Yaskawa INFORM job: long_pipe.JBI

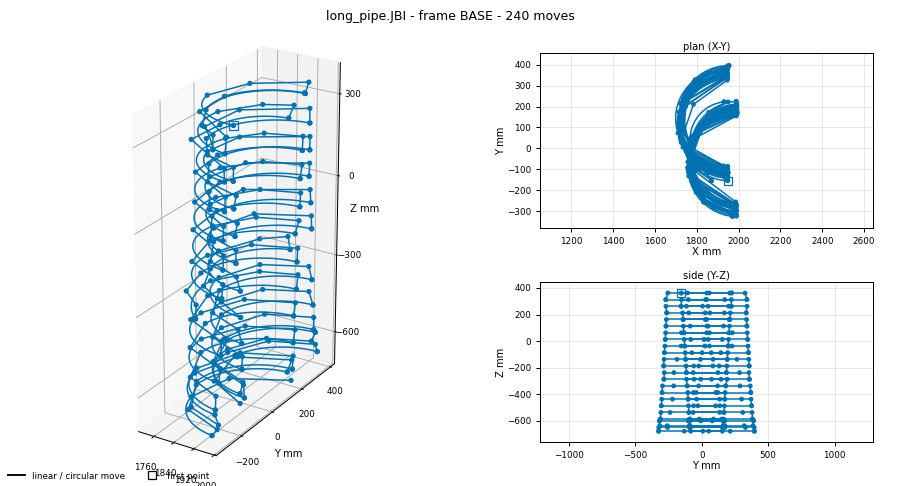
[picture p0: tool path of long_pipe.JBI in frame BASE, 240 of 346 moves have a stored position in this frame; points joined in program order, loops and branches not executed]
/JOB
//NAME long_pipe
//POS
///NPOS 336,0,336,0,0,0
///TOOL 0
///POSTYPE BASE
///RECTAN
///RCONF 0,0,0,0,0,0,0,0,0,0,0,0,0,0,0,0,0,0,0,0,0,0,0,0
C00000=1948.089852,-154.428104,361.796500,-91.436421,-90.000000,5.000000
C00001=1948.089852,-154.428104,361.796500,-91.436421,-90.000000,5.000000
C00002=1806.657138,-101.141800,361.796500,-121.772810,-90.000000,5.000000
C00003=1725.085960,37.670682,361.796500,-156.237975,-90.000000,5.000000
C00004=1725.085960,37.670682,361.796500,-156.237975,-90.000000,5.000000
C00005=1784.341244,210.221855,361.796500,157.427074,-90.000000,5.000000
C00006=1945.915028,325.931055,361.796500,92.921430,-89.999999,5.000000
C00007=1924.685573,339.998740,312.680000,98.705914,-90.000000,5.000000
C00008=1924.685573,339.998740,312.680000,98.705914,-90.000000,5.000000
C00009=1721.013871,191.051148,312.680000,167.503050,-90.000000,5.000000
C00010=1725.983821,28.850345,312.680000,-154.339335,-90.000000,5.000000
C00011=1725.983821,28.850345,312.680000,-154.339335,-90.000000,5.000000
C00012=1795.223122,-101.158175,312.680000,-123.700098,-90.000000,5.000000
C00013=1869.864544,-152.794566,312.680000,-106.341970,-90.000000,5.000000
C00014=1870.472685,-155.549095,262.680000,-106.088120,-90.000000,5.000000
C00015=1870.472685,-155.549095,262.680000,-106.088120,-90.000000,5.000000
C00016=1843.579568,-119.383824,262.680000,-113.403433,-90.000000,5.000000
C00017=1734.255940,6.180166,262.680000,-148.999232,-90.000000,5.000000
C00018=1734.255940,6.180166,262.680000,-148.999232,-90.000000,5.000000
C00019=1747.769146,201.411479,262.680000,163.296650,-90.000000,5.000000
C00020=1942.694355,340.824041,262.680000,93.618014,-90.000000,5.000000
C00021=1947.073941,334.429289,212.680000,92.455325,-90.000000,5.000000
C00022=1947.073941,334.429289,212.680000,92.455325,-90.000000,5.000000
C00023=1743.822934,197.595389,212.680000,164.546518,-90.000000,5.000000
C00024=1728.032875,25.819450,212.680000,-153.523098,-90.000000,5.000000
C00025=1728.032875,25.819450,212.680000,-153.523098,-90.000000,5.000000
C00026=1812.698059,-97.501858,212.680000,-121.105327,-90.000000,5.000000
C00027=1942.399423,-144.705270,212.680000,-92.632933,-90.000000,5.000000
C00028=1938.946956,-141.309317,162.680000,-93.368274,-90.000000,5.000000
C00029=1938.946956,-141.309317,162.680000,-93.368274,-90.000000,5.000000
C00030=1803.563456,-88.140401,162.680000,-123.759652,-89.999999,5.000000
C00031=1725.441837,36.442533,162.680000,-155.949661,-90.000000,5.000000
C00032=1725.441837,36.442533,162.680000,-155.949661,-90.000000,5.000000
C00033=1746.336332,205.754669,162.680000,162.318158,-90.000000,5.000000
C00034=1946.808055,337.053275,162.680000,92.499632,-90.000000,5.000000
C00035=1945.260351,339.688853,112.680000,92.907920,-89.999999,5.000000
C00036=1945.260351,339.688853,112.680000,92.907920,-89.999999,5.000000
C00037=1749.833887,217.231411,112.680000,159.191678,-90.000000,5.000000
C00038=1723.055881,48.584757,112.680000,-158.721498,-90.000000,5.000000
C00039=1723.055881,48.584757,112.680000,-158.721498,-90.000000,5.000000
C00040=1805.768560,-87.049483,112.680000,-123.500409,-90.000000,5.000000
C00041=1949.000324,-138.863334,112.680000,-91.329258,-90.000000,5.000000
C00042=1936.884281,-134.495510,62.680000,-93.882169,-90.000000,5.000000
C00043=1936.884281,-134.495510,62.680000,-93.882169,-90.000000,5.000000
C00044=1804.163203,-80.705374,62.680000,-124.539805,-89.999999,5.000000
C00045=1721.098993,58.361092,62.680000,-160.992048,-89.999999,5.000000
C00046=1721.098993,58.361092,62.680000,-160.992048,-89.999999,5.000000
C00047=1755.943683,229.421087,62.680000,155.640501,-90.000000,5.000000
C00048=1943.839534,342.441100,62.680000,93.267809,-89.999999,5.000000
C00049=1940.731812,345.123724,12.680000,94.086050,-90.000000,5.000000
C00050=1940.731812,345.123724,12.680000,94.086050,-90.000000,5.000000
C00051=1755.079974,233.890953,12.680000,154.680026,-90.000000,5.000000
C00052=1723.758836,48.110633,12.680000,-158.561082,-90.000000,5.000000
C00053=1723.758836,48.110633,12.680000,-158.561082,-90.000000,5.000000
C00054=1810.808406,-83.344167,12.680000,-123.034502,-89.999999,5.000000
C00055=1949.054836,-132.185836,12.680000,-91.350458,-90.000000,5.000000
C00056=1937.608440,-128.432526,-37.320000,-93.815495,-90.000000,5.000000
C00057=1937.608440,-128.432526,-37.320000,-93.815495,-90.000000,5.000000
C00058=1801.716874,-73.293020,-37.320000,-125.898714,-90.000000,5.000000
C00059=1721.874769,57.373947,-37.320000,-160.717445,-90.000000,5.000000
C00060=1721.874769,57.373947,-37.320000,-160.717445,-90.000000,5.000000
C00061=1748.048392,227.228459,-37.320000,156.976432,-90.000000,5.000000
C00062=1943.886424,348.166100,-37.320000,93.165704,-90.000000,5.000000
C00063=1945.403570,351.508515,-87.320000,92.707825,-90.000000,5.000000
C00064=1945.403570,351.508515,-87.320000,92.707825,-90.000000,5.000000
C00065=1764.794043,254.451315,-87.320000,148.823101,-90.000000,5.000000
C00066=1719.364469,71.495201,-87.320000,-164.022571,-90.000000,5.000000
C00067=1719.364469,71.495201,-87.320000,-164.022571,-90.000000,5.000000
C00068=1809.133318,-75.149384,-87.320000,-124.331343,-89.999999,5.000000
C00069=1938.729832,-125.214955,-87.320000,-93.619745,-89.999999,5.000000
C00070=1936.922427,-121.754242,-137.320000,-94.062838,-90.000000,5.000000
C00071=1936.922427,-121.754242,-137.320000,-94.062838,-90.000000,5.000000
C00072=1805.471154,-68.553083,-137.320000,-125.840133,-90.000000,5.000000
C00073=1717.543155,84.697835,-137.320000,-167.121689,-89.999999,5.000000
C00074=1717.543155,84.697835,-137.320000,-167.121689,-89.999999,5.000000
C00075=1769.057610,264.695420,-137.320000,146.025114,-90.000000,5.000000
C00076=1946.343505,354.471103,-137.320000,92.421083,-90.000000,5.000000
C00077=1946.850856,357.205562,-187.320000,92.257711,-90.000000,5.000000
C00078=1946.850856,357.205562,-187.320000,92.257711,-90.000000,5.000000
C00079=1769.073697,266.901665,-187.320000,145.558968,-90.000000,5.000000
C00080=1718.050928,83.425907,-187.320000,-166.803742,-90.000000,5.000000
C00081=1718.050928,83.425907,-187.320000,-166.803742,-90.000000,5.000000
C00082=1796.817162,-60.318135,-187.320000,-128.502754,-90.000000,5.000000
C00083=1936.521124,-118.597040,-187.320000,-94.201205,-90.000000,5.000000
C00084=1950.373259,-115.822362,-237.320000,-91.140926,-90.000000,5.000000
C00085=1950.373259,-115.822362,-237.320000,-91.140926,-90.000000,5.000000
C00086=1788.789474,-49.698601,-237.320000,-131.437564,-90.000000,5.000000
C00087=1713.556771,121.462071,-237.320000,-175.831712,-89.999999,5.000000
C00088=1713.556771,121.462071,-237.320000,-175.831712,-89.999999,5.000000
C00089=1779.676107,284.296664,-237.320000,140.440110,-89.999999,5.000000
C00090=1853.162637,354.889370,-237.320000,115.360721,-89.999999,5.000000
C00091=1860.386180,358.675829,-287.320000,113.409006,-90.000000,5.000000
C00092=1860.386180,358.675829,-287.320000,113.409006,-90.000000,5.000000
C00093=1730.946298,258.659756,-287.320000,151.960616,-89.999999,5.000000
C00094=1710.739488,73.262255,-287.320000,-164.943488,-89.999999,5.000000
C00095=1710.739488,73.262255,-287.320000,-164.943488,-89.999999,5.000000
C00096=1767.064394,-57.558684,-287.320000,-133.770440,-90.000000,5.000000
C00097=1859.771689,-115.665984,-287.320000,-110.584520,-90.000000,5.000000
C00098=1947.779730,-109.811027,-337.320000,-91.765092,-90.000000,5.000000
C00099=1947.779730,-109.811027,-337.320000,-91.765092,-90.000000,5.000000
C00100=1794.208585,-45.495626,-337.320000,-131.138093,-90.000000,5.000000
C00101=1715.967037,119.350089,-337.320000,-175.287684,-89.999999,5.000000
C00102=1715.967037,119.350089,-337.320000,-175.287684,-89.999999,5.000000
C00103=1779.362251,288.057746,-337.320000,139.769441,-89.999999,5.000000
C00104=1933.415288,364.951223,-337.320000,95.572089,-90.000000,5.000000
C00105=1944.191004,368.935356,-387.320000,92.804410,-90.000000,5.000000
C00106=1944.191004,368.935356,-387.320000,92.804410,-90.000000,5.000000
C00107=1776.821526,289.635713,-387.320000,139.876442,-90.000000,5.000000
C00108=1716.129048,121.164597,-387.320000,-175.716243,-89.999999,5.000000
C00109=1716.129048,121.164597,-387.320000,-175.716243,-89.999999,5.000000
C00110=1793.249925,-42.090790,-387.320000,-131.835982,-90.000000,5.000000
C00111=1934.966448,-105.589525,-387.320000,-94.785386,-89.999999,5.000000
C00112=1947.760101,-102.612541,-437.320000,-91.822275,-90.000000,5.000000
C00113=1947.760101,-102.612541,-437.320000,-91.822275,-90.000000,5.000000
C00114=1789.178214,-35.129272,-437.320000,-133.662724,-90.000000,5.000000
C00115=1715.792418,134.107597,-437.320000,-178.808772,-90.000000,5.000000
C00116=1715.792418,134.107597,-437.320000,-178.808772,-90.000000,5.000000
C00117=1783.843259,300.141568,-437.320000,136.817550,-90.000000,5.000000
C00118=1931.738733,371.088649,-437.320000,95.835639,-90.000000,5.000000
C00119=1946.586127,374.922161,-487.320000,92.152487,-89.999999,5.000000
C00120=1946.586127,374.922161,-487.320000,92.152487,-89.999999,5.000000
C00121=1781.433288,301.447997,-487.320000,136.985248,-90.000000,5.000000
C00122=1715.605097,135.687903,-487.320000,-179.187100,-90.000000,5.000000
C00123=1715.605097,135.687903,-487.320000,-179.187100,-90.000000,5.000000
C00124=1784.593790,-28.973026,-487.320000,-135.472019,-90.000000,5.000000
C00125=1948.352074,-100.171239,-487.320000,-91.699232,-90.000000,5.000000
C00126=1945.281183,-97.217812,-537.320000,-92.464026,-89.999999,5.000000
C00127=1945.281183,-97.217812,-537.320000,-92.464026,-89.999999,5.000000
C00128=1793.117537,-33.362696,-537.320000,-133.268365,-90.000000,5.000000
C00129=1716.145427,134.684238,-537.320000,-178.945025,-89.999999,5.000000
C00130=1716.145427,134.684238,-537.320000,-178.945025,-89.999999,5.000000
C00131=1787.067288,308.692942,-537.320000,134.793315,-90.000000,5.000000
C00132=1948.021952,378.690968,-537.320000,91.775708,-90.000000,5.000000
C00133=1947.011560,381.966547,-587.320000,91.989878,-90.000000,5.000000
C00134=1947.011560,381.966547,-587.320000,91.989878,-90.000000,5.000000
C00135=1789.216558,315.135500,-587.320000,133.358123,-90.000000,5.000000
C00136=1716.024354,149.961106,-587.320000,177.400513,-89.999999,5.000000
C00137=1716.024354,149.961106,-587.320000,177.400513,-89.999999,5.000000
C00138=1778.857613,-18.448199,-587.320000,-138.263643,-90.000000,5.000000
C00139=1947.332074,-94.134217,-587.320000,-91.993503,-90.000000,5.000000
C00140=1933.662341,-90.882022,-637.320000,-95.412052,-90.000000,5.000000
C00141=1933.662341,-90.882022,-637.320000,-95.412052,-90.000000,5.000000
C00142=1767.208531,-2.444827,-637.320000,-143.061065,-90.000000,5.000000
C00143=1716.921361,173.665472,-637.320000,171.752478,-89.999999,5.000000
C00144=1716.921361,173.665472,-637.320000,171.752478,-89.999999,5.000000
C00145=1789.055258,319.507135,-637.320000,132.684821,-90.000000,5.000000
C00146=1936.254340,385.591245,-637.320000,94.452796,-90.000000,5.000000
C00147=1949.256140,389.855264,-600.717460,180.000000,-60.000000,-88.585086
C00148=1949.256140,389.855264,-600.717460,180.000000,-60.000000,-88.585086
C00149=1796.012674,328.533492,-600.717460,180.000000,-60.000000,-49.915588
C00150=1716.317998,172.325490,-600.717460,180.000000,-60.000000,-7.912266
C00151=1716.317998,172.325490,-600.717460,180.000000,-60.000000,-7.912266
C00152=1775.299054,-8.028706,-600.717460,180.000000,-60.000000,39.236687
C00153=1946.064111,-89.050219,-600.717460,180.000000,-60.000000,87.644140
C00154=1948.372494,-86.795927,-650.717460,180.000000,-60.000000,88.205392
C00155=1948.372494,-86.795927,-650.717460,180.000000,-60.000000,88.205392
C00156=1775.279847,-6.023758,-650.717460,180.000000,-60.000000,38.849071
C00157=1716.545205,174.101681,-650.717460,180.000000,-60.000000,-8.337156
C00158=1716.545205,174.101681,-650.717460,180.000000,-60.000000,-8.337156
C00159=1792.571085,328.575973,-650.717460,-180.000000,-60.000000,-49.318058
C00160=1947.362979,394.502867,-650.717460,-180.000000,-60.000000,-88.186469
C00161=1954.969684,396.112738,-678.637460,-180.000000,-60.000000,-89.892927
C00162=1954.969684,396.112738,-678.637460,-180.000000,-60.000000,-89.892927
C00163=1803.482227,342.074602,-678.637460,-180.000000,-60.000000,-53.178896
C00164=1721.591344,214.572083,-678.637460,180.000000,-60.000000,-17.888195
C00165=1721.591344,214.572083,-678.637460,180.000000,-60.000000,-17.888195
C00166=1765.108221,8.381083,-678.637460,180.000000,-60.000000,34.477840
C00167=1929.576251,-83.832453,-678.637460,180.000000,-60.000000,83.379552
C00168=1988.723901,224.495613,362.682500,91.136861,-90.000000,5.000000
C00169=1988.723901,224.495613,362.682500,91.136861,-90.000000,5.000000
C00170=1851.653962,169.776784,362.682500,120.888805,-90.000000,5.000000
C00171=1780.186310,57.522696,362.682500,149.431820,-90.000000,5.000000
C00172=1780.186310,57.522696,362.682500,149.431820,-90.000000,5.000000
C00173=1789.875186,-107.742667,362.682500,-169.305957,-89.999999,5.000000
C00174=1986.239805,-255.786622,362.682500,-92.548667,-89.999999,5.000000
C00175=1990.121191,-271.036941,312.680000,-91.256333,-90.000000,5.000000
C00176=1990.121191,-271.036941,312.680000,-91.256333,-90.000000,5.000000
C00177=1808.253351,-148.428142,312.680000,-156.932564,-89.999999,5.000000
C00178=1767.408881,36.499458,312.680000,155.067828,-90.000000,5.000000
C00179=1767.408881,36.499458,312.680000,155.067828,-90.000000,5.000000
C00180=1857.792979,173.043612,312.680000,119.457652,-90.000000,5.000000
C00181=1950.206892,222.480952,312.680000,98.647445,-90.000000,5.000000
C00182=1930.045697,222.355400,262.680000,102.479797,-89.999999,5.000000
C00183=1930.045697,222.355400,262.680000,102.479797,-89.999999,5.000000
C00184=1817.772394,166.172520,262.680000,126.921293,-90.000000,5.000000
C00185=1768.075189,47.416654,262.680000,152.776908,-89.999999,5.000000
C00186=1768.075189,47.416654,262.680000,152.776908,-89.999999,5.000000
C00187=1760.588722,-115.433226,262.680000,-168.796077,-90.000000,5.000000
C00188=1985.937756,-270.370881,262.680000,-92.450043,-89.999999,5.000000
C00189=1983.203786,-264.021545,212.680000,-93.331225,-90.000000,5.000000
C00190=1983.203786,-264.021545,212.680000,-93.331225,-90.000000,5.000000
C00191=1778.387774,-96.104856,212.680000,-172.876660,-90.000000,5.000000
C00192=1781.359778,60.338071,212.680000,148.737810,-90.000000,5.000000
C00193=1781.359778,60.338071,212.680000,148.737810,-90.000000,5.000000
C00194=1865.910821,170.095672,212.680000,118.272216,-89.999999,5.000000
C00195=1990.964908,214.652948,212.680000,90.723891,-89.999999,5.000000
C00196=1990.361250,211.531002,162.680000,90.855171,-90.000000,5.000000
C00197=1990.361250,211.531002,162.680000,90.855171,-90.000000,5.000000
C00198=1855.009552,160.725264,162.680000,121.265397,-90.000000,5.000000
C00199=1771.949454,26.848917,162.680000,156.684157,-89.999999,5.000000
C00200=1771.949454,26.848917,162.680000,156.684157,-89.999999,5.000000
C00201=1792.474616,-139.695411,162.680000,-160.740769,-89.999999,5.000000
C00202=1988.687598,-266.951202,162.680000,-91.697121,-89.999999,5.000000
C00203=1986.544852,-269.556546,112.680000,-92.286765,-90.000000,5.000000
C00204=1986.544852,-269.556546,112.680000,-92.286765,-90.000000,5.000000
C00205=1788.365526,-135.956463,112.680000,-162.032162,-89.999999,5.000000
C00206=1774.573122,38.290928,112.680000,153.980638,-89.999999,5.000000
C00207=1774.573122,38.290928,112.680000,153.980638,-89.999999,5.000000
C00208=1865.058629,163.596407,112.680000,119.096094,-90.000000,5.000000
C00209=1991.745006,208.618149,112.680000,90.578695,-90.000000,5.000000
C00210=1987.652745,204.721634,62.680000,91.442958,-89.999999,5.000000
C00211=1987.652745,204.721634,62.680000,91.442958,-89.999999,5.000000
C00212=1860.097116,157.587789,62.680000,120.673992,-90.000000,5.000000
C00213=1774.256284,36.753283,62.680000,154.337162,-90.000000,5.000000
C00214=1774.256284,36.753283,62.680000,154.337162,-90.000000,5.000000
C00215=1797.219859,-153.509246,62.680000,-156.838660,-90.000000,5.000000
C00216=1985.392353,-272.459154,62.680000,-92.578281,-90.000000,5.000000
C00217=1983.896404,-274.918472,12.680000,-92.962976,-90.000000,5.000000
C00218=1983.896404,-274.918472,12.680000,-92.962976,-90.000000,5.000000
C00219=1802.598281,-166.501797,12.680000,-153.093322,-90.000000,5.000000
C00220=1769.911825,17.517256,12.680000,158.916075,-90.000000,5.000000
C00221=1769.911825,17.517256,12.680000,158.916075,-90.000000,5.000000
C00222=1860.434601,154.194398,12.680000,120.990949,-90.000000,5.000000
C00223=1991.728115,201.901968,12.680000,90.596607,-90.000000,5.000000
C00224=1990.844367,198.678738,-37.320000,90.792859,-89.999999,5.000000
C00225=1990.844367,198.678738,-37.320000,90.792859,-89.999999,5.000000
C00226=1848.887250,145.095727,-37.320000,124.218588,-90.000000,5.000000
C00227=1770.707112,23.440533,-37.320000,157.540917,-90.000000,5.000000
C00228=1770.707112,23.440533,-37.320000,157.540917,-90.000000,5.000000
C00229=1791.125725,-155.813653,-37.320000,-156.910761,-89.999999,5.000000
C00230=1987.626168,-278.204845,-37.320000,-91.896390,-90.000000,5.000000
C00231=1987.302870,-281.404691,-87.320000,-91.954979,-90.000000,5.000000
C00232=1987.302870,-281.404691,-87.320000,-91.954979,-90.000000,5.000000
C00233=1802.163860,-174.716993,-87.320000,-151.231840,-90.000000,5.000000
C00234=1766.018401,2.495406,-87.320000,162.607090,-90.000000,5.000000
C00235=1766.018401,2.495406,-87.320000,162.607090,-90.000000,5.000000
C00236=1852.133956,143.567440,-87.320000,123.809976,-90.000000,5.000000
C00237=1990.301803,195.483467,-87.320000,90.919903,-90.000000,5.000000
C00238=1978.075101,191.483388,-137.320000,93.617729,-90.000000,5.000000
C00239=1978.075101,191.483388,-137.320000,93.617729,-90.000000,5.000000
C00240=1840.480246,132.727671,-137.320000,127.358362,-89.999999,5.000000
C00241=1763.569258,-10.937979,-137.320000,165.868582,-90.000000,5.000000
C00242=1763.569258,-10.937979,-137.320000,165.868582,-90.000000,5.000000
C00243=1805.736775,-186.129334,-137.320000,-148.206757,-90.000000,5.000000
C00244=1988.495735,-284.497788,-137.320000,-91.609942,-90.000000,5.000000
C00245=1986.431281,-287.235224,-187.320000,-92.131405,-90.000000,5.000000
C00246=1986.431281,-287.235224,-187.320000,-92.131405,-90.000000,5.000000
C00247=1811.881725,-196.821195,-187.320000,-145.036956,-90.000000,5.000000
C00248=1761.960998,-22.671143,-187.320000,168.713269,-90.000000,5.000000
C00249=1761.960998,-22.671143,-187.320000,168.713269,-90.000000,5.000000
C00250=1841.420154,130.973540,-187.320000,127.430524,-89.999999,5.000000
C00251=1990.349923,189.068152,-187.320000,90.932082,-90.000000,5.000000
C00252=1990.050783,185.617204,-237.320000,91.011979,-90.000000,5.000000
C00253=1990.050783,185.617204,-237.320000,91.011979,-90.000000,5.000000
C00254=1834.684708,121.001254,-237.320000,130.063431,-89.999999,5.000000
C00255=1760.682694,-64.207382,-237.320000,178.803723,-90.000000,5.000000
C00256=1760.682694,-64.207382,-237.320000,178.803723,-90.000000,5.000000
C00257=1797.351101,-209.746240,-237.320000,-144.501034,-90.000000,5.000000
C00258=1883.887097,-282.491417,-237.320000,-117.409868,-90.000000,5.000000
C00259=1883.201806,-285.218759,-287.320000,-117.257350,-90.000000,5.000000
C00260=1883.201806,-285.218759,-287.320000,-117.257350,-90.000000,5.000000
C00261=1825.084107,-222.094242,-287.320000,-137.922519,-89.999999,5.000000
C00262=1764.084591,-8.534115,-287.320000,165.277808,-89.999999,5.000000
C00263=1764.084591,-8.534115,-287.320000,165.277808,-89.999999,5.000000
C00264=1865.504387,144.884540,-287.320000,121.093583,-90.000000,5.000000
C00265=1991.271457,191.290911,-287.320000,90.721389,-90.000000,5.000000
C00266=1992.213057,180.049202,-337.320000,90.537420,-89.999999,5.000000
C00267=1992.213057,180.049202,-337.320000,90.537420,-89.999999,5.000000
C00268=1842.768568,120.678380,-337.320000,128.653535,-90.000000,5.000000
C00269=1762.340076,-24.256685,-337.320000,169.071992,-90.000000,5.000000
C00270=1762.340076,-24.256685,-337.320000,169.071992,-90.000000,5.000000
C00271=1815.684610,-211.948344,-337.320000,-141.386116,-90.000000,5.000000
C00272=1990.619924,-295.785464,-337.320000,-90.993206,-90.000000,5.000000
C00273=1989.404799,-299.058471,-387.320000,-91.281699,-90.000000,5.000000
C00274=1989.404799,-299.058471,-387.320000,-91.281699,-90.000000,5.000000
C00275=1817.803991,-218.401001,-387.320000,-139.809827,-90.000000,5.000000
C00276=1759.664484,-62.758438,-387.320000,178.455668,-90.000000,5.000000
C00277=1759.664484,-62.758438,-387.320000,178.455668,-90.000000,5.000000
C00278=1828.364267,105.798466,-387.320000,133.538214,-90.000000,5.000000
C00279=1991.095267,175.932092,-387.320000,90.807795,-90.000000,5.000000
C00280=1986.677500,172.639516,-437.320000,91.865307,-90.000000,5.000000
C00281=1986.677500,172.639516,-437.320000,91.865307,-90.000000,5.000000
C00282=1838.667500,112.210894,-437.320000,130.688785,-90.000000,5.000000
C00283=1760.491814,-38.416294,-437.320000,172.533603,-89.999999,5.000000
C00284=1760.491814,-38.416294,-437.320000,172.533603,-89.999999,5.000000
C00285=1817.624442,-220.562088,-437.320000,-139.432211,-90.000000,5.000000
C00286=1987.883042,-301.728441,-437.320000,-91.641542,-90.000000,5.000000
C00287=1985.247473,-304.911428,-487.320000,-92.259004,-90.000000,5.000000
C00288=1985.247473,-304.911428,-487.320000,-92.259004,-90.000000,5.000000
C00289=1822.257694,-228.909254,-487.320000,-137.151015,-90.000000,5.000000
C00290=1759.212747,-61.758926,-487.320000,178.215493,-89.999999,5.000000
C00291=1759.212747,-61.758926,-487.320000,178.215493,-89.999999,5.000000
C00292=1833.533969,103.494646,-487.320000,133.013725,-89.999999,5.000000
C00293=1994.389046,170.058466,-487.320000,90.038562,-89.999999,5.000000
C00294=1988.965347,167.170212,-537.320000,91.354084,-90.000000,5.000000
C00295=1988.965347,167.170212,-537.320000,91.354084,-90.000000,5.000000
C00296=1829.253863,98.080224,-537.320000,134.676860,-90.000000,5.000000
C00297=1758.473988,-64.868502,-537.320000,178.975307,-89.999999,5.000000
C00298=1758.473988,-64.868502,-537.320000,178.975307,-89.999999,5.000000
C00299=1829.427702,-238.645140,-537.320000,-134.241324,-90.000000,5.000000
C00300=1975.364931,-308.234625,-537.320000,-94.586676,-90.000000,5.000000
C00301=1975.236574,-311.699949,-587.320000,-94.551559,-90.000000,5.000000
C00302=1975.236574,-311.699949,-587.320000,-94.551559,-90.000000,5.000000
C00303=1836.195005,-246.344507,-587.320000,-131.777011,-90.000000,5.000000
C00304=1758.737755,-89.666560,-587.320000,-175.013344,-90.000000,5.000000
C00305=1758.737755,-89.666560,-587.320000,-175.013344,-90.000000,5.000000
C00306=1822.516562,88.137068,-587.320000,137.574592,-90.000000,5.000000
C00307=1991.448854,164.508584,-587.320000,90.760584,-90.000000,5.000000
C00308=1990.175249,161.542422,-637.320000,91.086680,-90.000000,5.000000
C00309=1990.175249,161.542422,-637.320000,91.086680,-90.000000,5.000000
C00310=1823.837144,87.489601,-637.320000,137.472448,-89.999999,5.000000
C00311=1758.260695,-91.342142,-637.320000,-174.620375,-90.000000,5.000000
C00312=1758.260695,-91.342142,-637.320000,-174.620375,-90.000000,5.000000
C00313=1845.642521,-259.789406,-637.320000,-127.984615,-89.999999,5.000000
C00314=1990.075289,-316.298432,-637.320000,-91.037000,-90.000000,5.000000
C00315=1978.106023,-319.375296,-600.717460,180.000000,-60.000000,86.241001
C00316=1978.106023,-319.375296,-600.717460,180.000000,-60.000000,86.241001
C00317=1838.085731,-257.356845,-600.717460,180.000000,-60.000000,50.270655
C00318=1758.291580,-103.001000,-600.717460,-180.000000,-60.000000,8.167839
C00319=1758.291580,-103.001000,-600.717460,-180.000000,-60.000000,8.167839
C00320=1817.041118,78.408197,-600.717460,-180.000000,-60.000000,-39.724542
C00321=1989.068439,159.142556,-600.717460,180.000000,-60.000000,-88.624173
C00322=1973.216715,156.317083,-650.717460,180.000000,-60.000000,-84.593463
C00323=1973.216715,156.317083,-650.717460,180.000000,-60.000000,-84.593463
C00324=1819.168955,78.026603,-650.717460,180.000000,-60.000000,-39.991455
C00325=1757.442863,-93.095838,-650.717460,180.000000,-60.000000,5.780954
C00326=1757.442863,-93.095838,-650.717460,180.000000,-60.000000,5.780954
C00327=1832.580243,-257.616030,-650.717460,180.000000,-60.000000,49.332743
C00328=1990.311058,-324.522349,-650.717460,-180.000000,-60.000000,89.049251
C00329=1970.245915,-325.142816,-678.489460,180.000000,-60.000000,84.577808
C00330=1970.245915,-325.142816,-678.489460,180.000000,-60.000000,84.577808
C00331=1853.844206,-279.415467,-678.489460,180.000000,-60.000000,56.217717
C00332=1761.617376,-132.249138,-678.489460,180.000000,-60.000000,15.170617
C00333=1761.617376,-132.249138,-678.489460,180.000000,-60.000000,15.170617
C00334=1799.162341,52.520588,-678.489460,180.000000,-60.000000,-31.898622
C00335=1989.522356,154.791492,-678.489460,180.000000,-60.000000,-88.713547
///POSTYPE PULSE
///PULSE
EX00000=0
EX00001=92160
EX00002=184320
EX00003=276480
///POSTYPE PULSE
///PULSE
EC00000=0
EC00001=0
EC00002=0
EC00003=0
EC00004=0
EC00005=0
EC00006=0
EC00007=0
EC00008=0
EC00009=0
EC00010=0
EC00011=0
EC00012=0
EC00013=0
EC00014=0
EC00015=0
EC00016=0
EC00017=0
EC00018=0
EC00019=0
EC00020=0
EC00021=0
EC00022=0
EC00023=0
EC00024=0
EC00025=0
EC00026=0
EC00027=0
EC00028=0
EC00029=0
EC00030=0
EC00031=0
EC00032=0
EC00033=0
EC00034=0
EC00035=0
EC00036=0
EC00037=0
EC00038=0
EC00039=0
EC00040=0
EC00041=0
EC00042=0
EC00043=0
EC00044=0
EC00045=0
EC00046=0
EC00047=0
EC00048=0
EC00049=0
EC00050=0
EC00051=0
EC00052=0
EC00053=0
EC00054=0
EC00055=0
EC00056=0
EC00057=0
EC00058=0
EC00059=0
EC00060=0
EC00061=0
EC00062=0
EC00063=0
EC00064=0
EC00065=0
EC00066=0
EC00067=0
EC00068=0
EC00069=0
EC00070=0
EC00071=0
EC00072=0
EC00073=0
EC00074=0
EC00075=0
EC00076=0
EC00077=0
EC00078=0
EC00079=0
EC00080=0
EC00081=0
EC00082=0
EC00083=0
EC00084=0
EC00085=0
EC00086=0
EC00087=0
EC00088=0
EC00089=0
EC00090=0
EC00091=0
EC00092=0
EC00093=0
EC00094=0
EC00095=0
EC00096=0
EC00097=0
EC00098=0
EC00099=0
EC00100=0
EC00101=0
EC00102=0
EC00103=0
EC00104=0
EC00105=0
EC00106=0
EC00107=0
EC00108=0
EC00109=0
EC00110=0
EC00111=0
EC00112=0
EC00113=0
EC00114=0
EC00115=0
EC00116=0
EC00117=0
EC00118=0
EC00119=0
EC00120=0
EC00121=0
EC00122=0
EC00123=0
EC00124=0
EC00125=0
EC00126=0
EC00127=0
EC00128=0
EC00129=0
EC00130=0
EC00131=0
EC00132=0
EC00133=0
EC00134=0
EC00135=0
EC00136=0
EC00137=0
EC00138=0
EC00139=0
EC00140=0
EC00141=0
EC00142=0
EC00143=0
EC00144=0
EC00145=0
EC00146=0
EC00147=0
EC00148=0
EC00149=0
EC00150=0
EC00151=0
EC00152=0
EC00153=0
EC00154=0
EC00155=0
EC00156=0
EC00157=0
EC00158=0
EC00159=0
EC00160=0
EC00161=0
EC00162=0
EC00163=0
EC00164=0
EC00165=0
EC00166=0
EC00167=0
EC00168=184320
EC00169=184320
EC00170=184320
EC00171=184320
EC00172=184320
EC00173=184320
EC00174=184320
EC00175=184320
EC00176=184320
EC00177=184320
EC00178=184320
EC00179=184320
EC00180=184320
EC00181=184320
EC00182=184320
EC00183=184320
EC00184=184320
EC00185=184320
EC00186=184320
EC00187=184320
EC00188=184320
EC00189=184320
EC00190=184320
EC00191=184320
EC00192=184320
EC00193=184320
EC00194=184320
EC00195=184320
EC00196=184320
EC00197=184320
EC00198=184320
EC00199=184320
EC00200=184320
EC00201=184320
EC00202=184320
EC00203=184320
EC00204=184320
EC00205=184320
EC00206=184320
EC00207=184320
EC00208=184320
EC00209=184320
EC00210=184320
EC00211=184320
EC00212=184320
EC00213=184320
EC00214=184320
EC00215=184320
EC00216=184320
EC00217=184320
EC00218=184320
EC00219=184320
EC00220=184320
EC00221=184320
EC00222=184320
EC00223=184320
EC00224=184320
EC00225=184320
EC00226=184320
EC00227=184320
EC00228=184320
EC00229=184320
EC00230=184320
EC00231=184320
EC00232=184320
EC00233=184320
EC00234=184320
EC00235=184320
EC00236=184320
EC00237=184320
EC00238=184320
EC00239=184320
EC00240=184320
EC00241=184320
EC00242=184320
EC00243=184320
EC00244=184320
EC00245=184320
EC00246=184320
EC00247=184320
EC00248=184320
EC00249=184320
EC00250=184320
EC00251=184320
EC00252=184320
EC00253=184320
EC00254=184320
EC00255=184320
EC00256=184320
EC00257=184320
EC00258=184320
EC00259=184320
EC00260=184320
EC00261=184320
EC00262=184320
EC00263=184320
EC00264=184320
EC00265=184320
EC00266=184320
EC00267=184320
EC00268=184320
EC00269=184320
EC00270=184320
EC00271=184320
EC00272=184320
EC00273=184320
EC00274=184320
EC00275=184320
EC00276=184320
EC00277=184320
EC00278=184320
EC00279=184320
EC00280=184320
EC00281=184320
EC00282=184320
EC00283=184320
EC00284=184320
EC00285=184320
EC00286=184320
EC00287=184320
EC00288=184320
EC00289=184320
EC00290=184320
EC00291=184320
EC00292=184320
EC00293=184320
EC00294=184320
EC00295=184320
EC00296=184320
EC00297=184320
EC00298=184320
EC00299=184320
EC00300=184320
EC00301=184320
EC00302=184320
EC00303=184320
EC00304=184320
EC00305=184320
EC00306=184320
EC00307=184320
EC00308=184320
EC00309=184320
EC00310=184320
EC00311=184320
EC00312=184320
EC00313=184320
EC00314=184320
EC00315=184320
EC00316=184320
EC00317=184320
EC00318=184320
EC00319=184320
EC00320=184320
EC00321=184320
EC00322=184320
EC00323=184320
EC00324=184320
EC00325=184320
EC00326=184320
EC00327=184320
EC00328=184320
EC00329=184320
EC00330=184320
EC00331=184320
EC00332=184320
EC00333=184320
EC00334=184320
EC00335=184320
//INST
///DATE 2023/07/12 09:53
///ATTR SC,RW,RJ
////FRAME BASE
///GROUP1 RB1,ST1
NOP
MOVJ P009 EX000 VJ=15.00
MOVJ P009 VJ=15.00
MOVJ C00000 EC00000 VJ=15.0
CALL JOB:SPYON
MOVC C00001 EC00001 V=150.0
MOVC C00002 EC00002 V=150.0
MOVC C00003 EC00003 V=150.0
MOVC C00004 EC00004 V=150.0
MOVC C00005 EC00005 V=150.0
MOVC C00006 EC00006 V=150.0
MOVL C00007 EC00007 V=150.0
MOVC C00008 EC00008 V=150.0
MOVC C00009 EC00009 V=150.0
MOVC C00010 EC00010 V=150.0
MOVC C00011 EC00011 V=150.0
MOVC C00012 EC00012 V=150.0
MOVC C00013 EC00013 V=150.0
MOVL C00014 EC00014 V=150.0
MOVC C00015 EC00015 V=150.0
MOVC C00016 EC00016 V=150.0
MOVC C00017 EC00017 V=150.0
MOVC C00018 EC00018 V=150.0
MOVC C00019 EC00019 V=150.0
MOVC C00020 EC00020 V=150.0
MOVL C00021 EC00021 V=150.0
MOVC C00022 EC00022 V=150.0
MOVC C00023 EC00023 V=150.0
MOVC C00024 EC00024 V=150.0
MOVC C00025 EC00025 V=150.0
MOVC C00026 EC00026 V=150.0
MOVC C00027 EC00027 V=150.0
MOVL C00028 EC00028 V=150.0
MOVC C00029 EC00029 V=150.0
MOVC C00030 EC00030 V=150.0
MOVC C00031 EC00031 V=150.0
MOVC C00032 EC00032 V=150.0
MOVC C00033 EC00033 V=150.0
MOVC C00034 EC00034 V=150.0
MOVL C00035 EC00035 V=150.0
MOVC C00036 EC00036 V=150.0
MOVC C00037 EC00037 V=150.0
MOVC C00038 EC00038 V=150.0
MOVC C00039 EC00039 V=150.0
MOVC C00040 EC00040 V=150.0
MOVC C00041 EC00041 V=150.0
MOVL C00042 EC00042 V=150.0
MOVC C00043 EC00043 V=150.0
MOVC C00044 EC00044 V=150.0
MOVC C00045 EC00045 V=150.0
MOVC C00046 EC00046 V=150.0
MOVC C00047 EC00047 V=150.0
MOVC C00048 EC00048 V=150.0
MOVL C00049 EC00049 V=150.0
MOVC C00050 EC00050 V=150.0
MOVC C00051 EC00051 V=150.0
MOVC C00052 EC00052 V=150.0
MOVC C00053 EC00053 V=150.0
MOVC C00054 EC00054 V=150.0
MOVC C00055 EC00055 V=150.0
MOVL C00056 EC00056 V=150.0
MOVC C00057 EC00057 V=150.0
MOVC C00058 EC00058 V=150.0
MOVC C00059 EC00059 V=150.0
MOVC C00060 EC00060 V=150.0
MOVC C00061 EC00061 V=150.0
MOVC C00062 EC00062 V=150.0
MOVL C00063 EC00063 V=150.0
MOVC C00064 EC00064 V=150.0
MOVC C00065 EC00065 V=150.0
MOVC C00066 EC00066 V=150.0
MOVC C00067 EC00067 V=150.0
MOVC C00068 EC00068 V=150.0
MOVC C00069 EC00069 V=150.0
MOVL C00070 EC00070 V=150.0
MOVC C00071 EC00071 V=150.0
MOVC C00072 EC00072 V=150.0
MOVC C00073 EC00073 V=150.0
MOVC C00074 EC00074 V=150.0
MOVC C00075 EC00075 V=150.0
MOVC C00076 EC00076 V=150.0
MOVL C00077 EC00077 V=150.0
MOVC C00078 EC00078 V=150.0
MOVC C00079 EC00079 V=150.0
MOVC C00080 EC00080 V=150.0
MOVC C00081 EC00081 V=150.0
MOVC C00082 EC00082 V=150.0
MOVC C00083 EC00083 V=150.0
MOVL C00084 EC00084 V=150.0
MOVC C00085 EC00085 V=150.0
MOVC C00086 EC00086 V=150.0
MOVC C00087 EC00087 V=150.0
MOVC C00088 EC00088 V=150.0
MOVC C00089 EC00089 V=150.0
MOVC C00090 EC00090 V=150.0
MOVL C00091 EC00091 V=150.0
MOVC C00092 EC00092 V=150.0
MOVC C00093 EC00093 V=150.0
MOVC C00094 EC00094 V=150.0
MOVC C00095 EC00095 V=150.0
MOVC C00096 EC00096 V=150.0
MOVC C00097 EC00097 V=150.0
MOVL C00098 EC00098 V=150.0
MOVC C00099 EC00099 V=150.0
MOVC C00100 EC00100 V=150.0
MOVC C00101 EC00101 V=150.0
MOVC C00102 EC00102 V=150.0
MOVC C00103 EC00103 V=150.0
MOVC C00104 EC00104 V=150.0
MOVL C00105 EC00105 V=150.0
MOVC C00106 EC00106 V=150.0
MOVC C00107 EC00107 V=150.0
MOVC C00108 EC00108 V=150.0
MOVC C00109 EC00109 V=150.0
MOVC C00110 EC00110 V=150.0
MOVC C00111 EC00111 V=150.0
MOVL C00112 EC00112 V=150.0
MOVC C00113 EC00113 V=150.0
MOVC C00114 EC00114 V=150.0
MOVC C00115 EC00115 V=150.0
MOVC C00116 EC00116 V=150.0
MOVC C00117 EC00117 V=150.0
MOVC C00118 EC00118 V=150.0
MOVL C00119 EC00119 V=150.0
MOVC C00120 EC00120 V=150.0
MOVC C00121 EC00121 V=150.0
MOVC C00122 EC00122 V=150.0
MOVC C00123 EC00123 V=150.0
MOVC C00124 EC00124 V=150.0
MOVC C00125 EC00125 V=150.0
MOVL C00126 EC00126 V=150.0
MOVC C00127 EC00127 V=150.0
MOVC C00128 EC00128 V=150.0
MOVC C00129 EC00129 V=150.0
MOVC C00130 EC00130 V=150.0
MOVC C00131 EC00131 V=150.0
MOVC C00132 EC00132 V=150.0
MOVL C00133 EC00133 V=150.0
MOVC C00134 EC00134 V=150.0
MOVC C00135 EC00135 V=150.0
MOVC C00136 EC00136 V=150.0
MOVC C00137 EC00137 V=150.0
MOVC C00138 EC00138 V=150.0
MOVC C00139 EC00139 V=150.0
MOVL C00140 EC00140 V=150.0
MOVC C00141 EC00141 V=150.0
MOVC C00142 EC00142 V=150.0
MOVC C00143 EC00143 V=150.0
MOVC C00144 EC00144 V=150.0
MOVC C00145 EC00145 V=150.0
MOVC C00146 EC00146 V=150.0
MOVL C00147 EC00147 V=150.0
MOVC C00148 EC00148 V=150.0
MOVC C00149 EC00149 V=150.0
MOVC C00150 EC00150 V=150.0
MOVC C00151 EC00151 V=150.0
MOVC C00152 EC00152 V=150.0
MOVC C00153 EC00153 V=150.0
MOVL C00154 EC00154 V=150.0
MOVC C00155 EC00155 V=150.0
MOVC C00156 EC00156 V=150.0
MOVC C00157 EC00157 V=150.0
MOVC C00158 EC00158 V=150.0
MOVC C00159 EC00159 V=150.0
MOVC C00160 EC00160 V=150.0
MOVL C00161 EC00161 V=150.0
MOVC C00162 EC00162 V=150.0
MOVC C00163 EC00163 V=150.0
MOVC C00164 EC00164 V=150.0
MOVC C00165 EC00165 V=150.0
MOVC C00166 EC00166 V=150.0
MOVC C00167 EC00167 V=150.0
CALL JOB:SPYOF
MOVJ P009 VJ=15.00
MOVL P009 EX00000 V=150.0
MOVJ P009 VJ=15.00
MOVL P009 EX00001 V=150.0
MOVJ C00168 EC00168 VJ=15.0
CALL JOB:SPYON
MOVC C00169 EC00169 V=150.0
MOVC C00170 EC00170 V=150.0
MOVC C00171 EC00171 V=150.0
MOVC C00172 EC00172 V=150.0
MOVC C00173 EC00173 V=150.0
MOVC C00174 EC00174 V=150.0
MOVL C00175 EC00175 V=150.0
MOVC C00176 EC00176 V=150.0
MOVC C00177 EC00177 V=150.0
MOVC C00178 EC00178 V=150.0
MOVC C00179 EC00179 V=150.0
MOVC C00180 EC00180 V=150.0
MOVC C00181 EC00181 V=150.0
MOVL C00182 EC00182 V=150.0
MOVC C00183 EC00183 V=150.0
MOVC C00184 EC00184 V=150.0
MOVC C00185 EC00185 V=150.0
MOVC C00186 EC00186 V=150.0
MOVC C00187 EC00187 V=150.0
MOVC C00188 EC00188 V=150.0
MOVL C00189 EC00189 V=150.0
MOVC C00190 EC00190 V=150.0
MOVC C00191 EC00191 V=150.0
MOVC C00192 EC00192 V=150.0
MOVC C00193 EC00193 V=150.0
MOVC C00194 EC00194 V=150.0
MOVC C00195 EC00195 V=150.0
MOVL C00196 EC00196 V=150.0
MOVC C00197 EC00197 V=150.0
MOVC C00198 EC00198 V=150.0
MOVC C00199 EC00199 V=150.0
MOVC C00200 EC00200 V=150.0
MOVC C00201 EC00201 V=150.0
MOVC C00202 EC00202 V=150.0
MOVL C00203 EC00203 V=150.0
MOVC C00204 EC00204 V=150.0
MOVC C00205 EC00205 V=150.0
MOVC C00206 EC00206 V=150.0
MOVC C00207 EC00207 V=150.0
MOVC C00208 EC00208 V=150.0
MOVC C00209 EC00209 V=150.0
MOVL C00210 EC00210 V=150.0
MOVC C00211 EC00211 V=150.0
MOVC C00212 EC00212 V=150.0
MOVC C00213 EC00213 V=150.0
MOVC C00214 EC00214 V=150.0
MOVC C00215 EC00215 V=150.0
MOVC C00216 EC00216 V=150.0
MOVL C00217 EC00217 V=150.0
MOVC C00218 EC00218 V=150.0
MOVC C00219 EC00219 V=150.0
MOVC C00220 EC00220 V=150.0
MOVC C00221 EC00221 V=150.0
MOVC C00222 EC00222 V=150.0
MOVC C00223 EC00223 V=150.0
MOVL C00224 EC00224 V=150.0
MOVC C00225 EC00225 V=150.0
MOVC C00226 EC00226 V=150.0
MOVC C00227 EC00227 V=150.0
MOVC C00228 EC00228 V=150.0
MOVC C00229 EC00229 V=150.0
MOVC C00230 EC00230 V=150.0
MOVL C00231 EC00231 V=150.0
MOVC C00232 EC00232 V=150.0
MOVC C00233 EC00233 V=150.0
MOVC C00234 EC00234 V=150.0
MOVC C00235 EC00235 V=150.0
MOVC C00236 EC00236 V=150.0
MOVC C00237 EC00237 V=150.0
MOVL C00238 EC00238 V=150.0
MOVC C00239 EC00239 V=150.0
MOVC C00240 EC00240 V=150.0
MOVC C00241 EC00241 V=150.0
MOVC C00242 EC00242 V=150.0
MOVC C00243 EC00243 V=150.0
MOVC C00244 EC00244 V=150.0
MOVL C00245 EC00245 V=150.0
MOVC C00246 EC00246 V=150.0
MOVC C00247 EC00247 V=150.0
MOVC C00248 EC00248 V=150.0
MOVC C00249 EC00249 V=150.0
MOVC C00250 EC00250 V=150.0
MOVC C00251 EC00251 V=150.0
MOVL C00252 EC00252 V=150.0
MOVC C00253 EC00253 V=150.0
MOVC C00254 EC00254 V=150.0
MOVC C00255 EC00255 V=150.0
MOVC C00256 EC00256 V=150.0
MOVC C00257 EC00257 V=150.0
MOVC C00258 EC00258 V=150.0
MOVL C00259 EC00259 V=150.0
MOVC C00260 EC00260 V=150.0
MOVC C00261 EC00261 V=150.0
MOVC C00262 EC00262 V=150.0
MOVC C00263 EC00263 V=150.0
MOVC C00264 EC00264 V=150.0
MOVC C00265 EC00265 V=150.0
MOVL C00266 EC00266 V=150.0
MOVC C00267 EC00267 V=150.0
MOVC C00268 EC00268 V=150.0
MOVC C00269 EC00269 V=150.0
MOVC C00270 EC00270 V=150.0
MOVC C00271 EC00271 V=150.0
MOVC C00272 EC00272 V=150.0
MOVL C00273 EC00273 V=150.0
MOVC C00274 EC00274 V=150.0
MOVC C00275 EC00275 V=150.0
MOVC C00276 EC00276 V=150.0
MOVC C00277 EC00277 V=150.0
MOVC C00278 EC00278 V=150.0
MOVC C00279 EC00279 V=150.0
MOVL C00280 EC00280 V=150.0
MOVC C00281 EC00281 V=150.0
MOVC C00282 EC00282 V=150.0
MOVC C00283 EC00283 V=150.0
MOVC C00284 EC00284 V=150.0
MOVC C00285 EC00285 V=150.0
MOVC C00286 EC00286 V=150.0
MOVL C00287 EC00287 V=150.0
MOVC C00288 EC00288 V=150.0
MOVC C00289 EC00289 V=150.0
MOVC C00290 EC00290 V=150.0
MOVC C00291 EC00291 V=150.0
MOVC C00292 EC00292 V=150.0
MOVC C00293 EC00293 V=150.0
MOVL C00294 EC00294 V=150.0
MOVC C00295 EC00295 V=150.0
MOVC C00296 EC00296 V=150.0
MOVC C00297 EC00297 V=150.0
MOVC C00298 EC00298 V=150.0
MOVC C00299 EC00299 V=150.0
MOVC C00300 EC00300 V=150.0
MOVL C00301 EC00301 V=150.0
MOVC C00302 EC00302 V=150.0
MOVC C00303 EC00303 V=150.0
MOVC C00304 EC00304 V=150.0
MOVC C00305 EC00305 V=150.0
MOVC C00306 EC00306 V=150.0
MOVC C00307 EC00307 V=150.0
MOVL C00308 EC00308 V=150.0
MOVC C00309 EC00309 V=150.0
MOVC C00310 EC00310 V=150.0
MOVC C00311 EC00311 V=150.0
MOVC C00312 EC00312 V=150.0
MOVC C00313 EC00313 V=150.0
MOVC C00314 EC00314 V=150.0
MOVL C00315 EC00315 V=150.0
MOVC C00316 EC00316 V=150.0
MOVC C00317 EC00317 V=150.0
MOVC C00318 EC00318 V=150.0
MOVC C00319 EC00319 V=150.0
MOVC C00320 EC00320 V=150.0
MOVC C00321 EC00321 V=150.0
MOVL C00322 EC00322 V=150.0
MOVC C00323 EC00323 V=150.0
MOVC C00324 EC00324 V=150.0
MOVC C00325 EC00325 V=150.0
MOVC C00326 EC00326 V=150.0
MOVC C00327 EC00327 V=150.0
MOVC C00328 EC00328 V=150.0
MOVL C00329 EC00329 V=150.0
MOVC C00330 EC00330 V=150.0
MOVC C00331 EC00331 V=150.0
MOVC C00332 EC00332 V=150.0
MOVC C00333 EC00333 V=150.0
MOVC C00334 EC00334 V=150.0
MOVC C00335 EC00335 V=150.0
CALL JOB:SPYOF
MOVJ P009 VJ=15.00
MOVL P009 EX00002 V=150.0
MOVJ P009 VJ=15.00
MOVL P009 EX00003 V=150.0
END
